{attribute 'linkalways'} 
{attribute 'no_explicit_call' := 'This FB is a CLASS and must be accessed using methods or properties'}
{attribute 'enable_dynamic_creation'}
FUNCTION_BLOCK Node_F_VN_AppendToContainer_TcVnVector4_USINT EXTENDS VisionNode
VAR
    aElement : _TcVnVector4_USINT;
    ipContainer : _ITcVnContainer;
    hrPrev : _HRESULT(S_OK);
	hresult : _HRESULT(S_OK);
END_VAR

METHOD PUBLIC  Clone : I_Node
VAR
	pNode : POINTER TO Node_F_VN_AppendToContainer_TcVnVector4_USINT;
END_VAR
pNode := __NEW(Node_F_VN_AppendToContainer_TcVnVector4_USINT);
Clone := pNode^;
END_METHOD

METHOD FB_init : BOOL
VAR_INPUT
	bInitRetains : BOOL; // if TRUE, the retain variables are initialized (warm start / cold start)
	bInCopyCode : BOOL;  // if TRUE, the instance afterwards gets moved into the copy code (online change)
END_VAR
AddInput('aElement', aElement);
AddInput('ipContainer', ipContainer);
AddInput('hrPrev', hrPrev);
AddOutput('ipContainer', ipContainer);
AddOutput('hresult',hresult);
END_METHOD

METHOD PROTECTED OnExecute : HRESULT
hresult.Value := F_VN_AppendToContainer_TcVnVector4_USINT(
    aElement := aElement.Value,
	ipContainer := ipContainer.Value,
	hrPrev:= hrPrev.Value);
END_METHOD

METHOD PUBLIC PreExecutionCheck
VAR_INPUT
	Check : I_PreExecutionChecks;
END_VAR
Check.IsTrue(ipContainer.IsValid, 'ipContainer must be a valid container');
END_METHOD

END_FUNCTION_BLOCK

(* stored: Version 1.1.0.1, ProductVersion 3.1.4024.13
   POU Node_F_VN_AppendToContainer_TcVnVector4_USINT: Id {2d84b52e-0e0e-4502-afbe-a1653a396d6f}, SpecialFunc None
   Folder Constructor: Id {b17a9dcd-b9f3-4c94-8b79-67139c474bca}
   Method Clone: Id {fbc6a51e-344b-4289-9c8b-3d2b4d57c3ba}
   Method FB_init: Id {465adcae-8d63-4d36-b33e-0d1f9d87f8fc}
   Method OnExecute: Id {9c6ab20e-ed80-4a31-8bfa-fee3ff98f1ee}
   Method PreExecutionCheck: Id {76f9c600-c776-4836-a695-909a1afe5826} *)
